(*
SPDX-FileCopyrightText: © 2026 Oleksandr Tiutyk <trofimich@gmail.com>
SPDX-License-Identifier: MIT
License: https://opensource.org/license/mit
*)

(*!
<summary>Provides common automation state, diagnostics and local event reception.</summary>
<description>
Both event delivery directions call OnEventReceived locally. Descendants with a parent or children extend the
appropriate direction with forwarding; terminal nodes only receive the event. Event delivery is synchronous
and borrowed, without retaining the event or transferring ownership. Delivery and forwarding are independent
of Enabled and operational state. OnEventReceived decides whether the component should react in its current
state; inactivity alone does not stop propagation. The event must be non-null and live. Handler exceptions
abort delivery and propagate to the caller; effects of handlers already invoked are not rolled back.
Initialization validates required dependencies before hooks. Child types require a live borrowed parent.
FALSE reports pending initialization or failure; INVALID must never report successful initialization.
Error and HasError observe the same diagnostic selected by GetReportedError(). The base exposes its execution error.
Required error snapshots precede logging callbacks so they preserve the primary diagnostic.
Stop transitions a WORKING component (and, for branches, all WORKING children) to STOPPED regardless of
Enabled, so a runtime stop reaction also stops a disabled working component and preserves its Reset requirement.
</description>
*)

FUNCTION_BLOCK ABSTRACT AutomationComponent EXTENDS TOF_Core.Object IMPLEMENTS IAutomationComponent
VAR
	{attribute 'hide'} 
	_Name : WSTRING;

	{attribute 'hide'} 
	_Enabled : BOOL := TRUE;
	
	{attribute 'hide'} 
	_OperationalState : OPERATIONAL_STATE;
	//! <summary>Counts state transitions so output traversal can detect a stop followed by an immediate reset.</summary>
	_OperationalStateRevision : UDINT;	
	{attribute 'hide'} 
	_OperationalStateReason : WSTRING(255);	

	_InitializationTimer : Tc2_Standard.TON;
	
	{attribute 'hide'} 
	_Error : TOF_Core.ERROR;
	
	{attribute 'hide'} 
	_ExceptionHandlingPolicy : TOF_Core.IExceptionHandlingPolicy;
END_VAR

(*!
<summary>Receives a broadcast event locally without forwarding it.</summary>
<description>
Calls OnEventReceived once. This is the terminal behavior for a leaf; branches override it to forward to
children unless propagation is stopped. Handled does not suppress delivery. The event is borrowed for this
synchronous call and is not retained or owned by the component.
</description>
*)

METHOD BroadcastEvent
VAR_INPUT
	event : TOF_Core.IEvent;
END_VAR
VAR
	stopPropagation : BOOL;
END_VAR
OnEventReceived(event := event, stopPropagation => stopPropagation);
END_METHOD

(*!
<summary>Receives a bubbling event locally without forwarding it.</summary>
<description>
Calls OnEventReceived once. This is the terminal behavior for a root; components with a parent override it to
forward upward unless propagation is stopped. Handled does not suppress delivery. The event is borrowed for
this synchronous call and is not retained or owned by the component.
</description>
*)

METHOD BubbleEvent
VAR_INPUT
	event : TOF_Core.IEvent;
END_VAR
VAR
	stopPropagation : BOOL;
END_VAR
OnEventReceived(event := event, stopPropagation => stopPropagation);
END_METHOD

(*!
<summary>Disables cyclic execution and invokes disable hooks.</summary>
<description>
Branches also disable their children. Hook exceptions propagate to the caller without rolling back prior
effects.
</description>
*)
METHOD ABSTRACT Disable
END_METHOD

(*!
<summary>Enables cyclic execution and invokes enable hooks.</summary>
<description>
Enabling does not automatically reset a STOPPED component; components stopped while disabled or disabled
while stopped remain STOPPED after Enable until explicitly Reset.
</description>
<param name="includeChildren">When TRUE on a branch, recursively enables child components.</param>
*)
METHOD ABSTRACT Enable
VAR_INPUT
	includeChildren : BOOL := TRUE;
END_VAR
END_METHOD

{attribute 'monitoring' := 'call'}
PROPERTY FINAL Enabled : BOOL
GET
Enabled := _Enabled;
END_GET
END_PROPERTY

(*!
<summary>Gets a borrowed view of the currently reported diagnostic.</summary>
<description>
Read the property again after component execution because a descendant can select a different record.
Observe the reference on the owning task while the component is live, following the IErrorProvider contract.
</description>
*)
{attribute 'monitoring' := 'call'}
PROPERTY FINAL Error : REFERENCE TO TOF_Core.ERROR
GET
Error REF= GetReportedError();
END_GET
END_PROPERTY

{attribute 'monitoring' := 'call'}
PROPERTY FINAL ExceptionHandlingPolicy : TOF_Core.IExceptionHandlingPolicy
GET
ExceptionHandlingPolicy := _ExceptionHandlingPolicy;
END_GET
SET
_ExceptionHandlingPolicy := ExceptionHandlingPolicy;
END_SET
END_PROPERTY

METHOD ABSTRACT Execute
END_METHOD

METHOD FB_init : BOOL
VAR_INPUT
	bInitRetains : BOOL; // TRUE: the retain variables are initialized (reset warm / reset cold)
	bInCopyCode : BOOL;  // TRUE: the instance will be copied to the copy code afterward (online change)
	name : WSTRING;
END_VAR
_Name := SEL(
	TOF_Core.WideStrings.IsNullOrWhiteSpace(stringToCheck := name),
	name,
	GetDefaultName()
);
_InitializationTimer.PT := Parameters.InitializationTimeout;
END_METHOD

METHOD FINAL GetEffectiveExceptionHandlingPolicy : TOF_Core.IExceptionHandlingPolicy
VAR
	thisAsChildAutomationComponent : IChildAutomationComponent;
	parent : IParentAutomationComponent;
END_VAR
IF _ExceptionHandlingPolicy <> 0 THEN
	GetEffectiveExceptionHandlingPolicy := _ExceptionHandlingPolicy;
ELSIF __QUERYINTERFACE(THIS^, thisAsChildAutomationComponent) THEN
	parent := thisAsChildAutomationComponent.Parent;

	IF parent <> 0 THEN
		GetEffectiveExceptionHandlingPolicy := parent.GetEffectiveExceptionHandlingPolicy();
	END_IF
END_IF
END_METHOD

METHOD PROTECTED FINAL GetErrorSeverityByExceptionReaction : TOF_Core.ERROR_SEVERITY
VAR_INPUT
	exceptionReaction : TOF_Core.EXCEPTION_REACTION;
END_VAR
IF exceptionReaction = TOF_Core.EXCEPTION_REACTION.SET_ERROR_AND_STOP THEN
	GetErrorSeverityByExceptionReaction := TOF_Core.ERROR_SEVERITY.CRITICAL;
ELSE
	GetErrorSeverityByExceptionReaction := TOF_Core.ERROR_SEVERITY.ERROR;
END_IF
END_METHOD

(*!
<summary>Prepares diagnostic text locally before passing it to read-only logging or exception parameters.</summary>
<description>Computed diagnostic strings are held in local buffers for the duration of the receiving call.</description>
*)
METHOD HandleRequest
VAR_INPUT
	request	: TOF_Core.INamed;
END_VAR
VAR
	formattedLogMessage : TOF_Core.ERROR_MESSAGE;
END_VAR
IF request = 0 THEN
	RETURN;
END_IF

formattedLogMessage := TOF_Core.WideStrings.Concat255("Request ", request.Name, " was not handled");

TOF_Core.LogManager.TryLogMessage(
	message := formattedLogMessage,
	category := TOF_Core.LOG_CATEGORY.INFORMATION,
	topic1 := TO_WSTRING(ClassName),
	topic2 := TO_WSTRING(__POUNAME())
);
END_METHOD

(*!
<summary>Selects the live diagnostic record exposed by Error and HasError.</summary>
<description>
Returns the component's execution record by default. An override must return a valid reference to
instance-owned storage, including when no error is active. Selection must be side-effect free and must
complete without exceptions. Read the selected record on the component's owner task.
</description>
*)
METHOD PROTECTED GetReportedError : REFERENCE TO TOF_Core.ERROR
GetReportedError REF= _Error;
END_METHOD

(*!
<summary>Reports whether the currently selected diagnostic contains an active error.</summary>
*)
{attribute 'monitoring' := 'call'}
PROPERTY FINAL HasError : BOOL
GET
HasError := THIS^.Error.HasError;
END_GET
END_PROPERTY

(*!
<summary>Sets the maximum wait for pending initialization.</summary>
<description>
T#0S selects Parameters.InitializationTimeout immediately upon assignment, so the getter always returns the
active non-zero duration. Branches expand this duration to at least the maximum InitializationTimeout of their
children during initialization.
</description>
*)
{attribute 'monitoring' := 'call'}
PROPERTY FINAL InitializationTimeout : TIME
GET
InitializationTimeout := _InitializationTimer.PT;
END_GET
SET
_InitializationTimer.PT := SEL(
	InitializationTimeout = T#0S,
	InitializationTimeout,
	Parameters.InitializationTimeout
);
END_SET
END_PROPERTY

(*!
<summary>Validates mandatory dependencies and advances initialization.</summary>
<description>
FALSE reports pending work or failure. An INVALID component must never report TRUE. Caught failures
record a critical copied error and enter terminal INVALID. Completed callback effects are not rolled back.
Only a pending call evaluates the timeout. Completion on the deadline cycle succeeds.
</description>
*)
METHOD ABSTRACT Initialize : BOOL
END_METHOD

{attribute 'monitoring' := 'call'}
PROPERTY FINAL Name : REFERENCE TO WSTRING
GET
Name REF= _Name;
END_GET
END_PROPERTY

(*!
<summary>Handles a delivered event locally and can stop further propagation along the current route.</summary>
<description>
May be called regardless of Enabled or operational state, including while disabled or stopped. The handler
checks state when its reaction requires it. Ignoring an event does not stop propagation; leave stopPropagation
FALSE unless further delivery along the route must be stopped. The event must be non-null and live and is
borrowed only for the call; do not retain it for later use. Handled and stopPropagation are independent.
Setting stopPropagation stops bubbling to the parent or broadcasting into this node's descendants; it does not
cancel sibling branches in the caller. An exception aborts delivery and propagates to the dispatch caller,
without rolling back prior effects.
</description>
*)

METHOD OnEventReceived
VAR_INPUT
	event : TOF_Core.IEvent;
END_VAR
VAR_OUTPUT
	stopPropagation : BOOL;
END_VAR
END_METHOD

METHOD PROTECTED FINAL OnHandleException : TOF_Core.EXCEPTION_REACTION
VAR_INPUT
	exception : TOF_Core.IException;
	failedMethodName : STRING(255);
END_VAR
VAR
	effectiveExceptionHandlingPolicy : TOF_Core.IExceptionHandlingPolicy;
END_VAR
effectiveExceptionHandlingPolicy := GetEffectiveExceptionHandlingPolicy();

IF effectiveExceptionHandlingPolicy <> 0 THEN
	OnHandleException := effectiveExceptionHandlingPolicy.HandleException(
		exception := exception,
		handlingObject := THIS^,
		failedMethodName := failedMethodName
	);
ELSE
	OnHandleException := TOF_Core.EXCEPTION_REACTION.SET_ERROR_AND_STOP;
END_IF
END_METHOD

METHOD PROTECTED OnOperationalStateChanged
VAR_INPUT
	previousState : OPERATIONAL_STATE;
END_VAR
END_METHOD

(*!
<summary>Runs at the start of cyclic working execution when clearing a non-critical error.</summary>
<description>
The base implementation does nothing. An exception raised by OnRecover always records a copied CRITICAL
error and stops the component without consulting ExceptionHandlingPolicy.
</description>
*)
METHOD PROTECTED OnRecover
END_METHOD

{attribute 'monitoring' := 'call'}
PROPERTY FINAL OperationalState : OPERATIONAL_STATE
GET
OperationalState := _OperationalState;
END_GET
END_PROPERTY

{attribute 'monitoring' := 'call'}
PROPERTY FINAL OperationalStateReason : REFERENCE TO WSTRING(255)
GET
OperationalStateReason REF= _OperationalStateReason;
END_GET
END_PROPERTY

METHOD PROTECTED ProcessChildError
VAR_INPUT
	childError : REFERENCE TO TOF_Core.ERROR;  
	childErrorReaction : CHILD_CRITICAL_ERROR_REACTION;	
	childErrorSourceHint : WSTRING(255);
END_VAR

IF NOT __ISVALIDREF(childError)
	OR_ELSE childError.Empty
	OR_ELSE childError.Severity <> TOF_Core.ERROR_SEVERITY.CRITICAL
THEN
	RETURN;
END_IF

IF OperationalState <> OPERATIONAL_STATE.INITIALIZING THEN
	CASE childErrorReaction OF
		CHILD_CRITICAL_ERROR_REACTION.SET_ERROR_AND_CONTINUE:
			IF _Error.Empty THEN
				_Error := childError;
				_Error.SetSeverity(severity := TOF_Core.ERROR_SEVERITY.ERROR);
			END_IF		
		
		CHILD_CRITICAL_ERROR_REACTION.SET_ERROR_AND_STOP:
			IF _Error.Empty OR_ELSE _Error.Severity < TOF_Core.ERROR_SEVERITY.CRITICAL THEN
				_Error := childError;
				_Error.SetSeverity(severity := TOF_Core.ERROR_SEVERITY.CRITICAL);
			END_IF	
			
			IF OperationalState = OPERATIONAL_STATE.WORKING THEN
				Stop(reason := childErrorSourceHint);		
			END_IF
	END_CASE
ELSE
	_Error := childError;
	
	SetOperationalState(state := OPERATIONAL_STATE.INVALID, reason := childErrorSourceHint);		
END_IF
END_METHOD

(*!
<summary>Applies an exception reaction to copied diagnostics and operational state.</summary>
<description>
Initialization failures enter INVALID with a critical error. At runtime a stop reaction records a
critical error and calls Stop on a working component, including when disabled (since Stop transitions
WORKING components and WORKING children to STOPPED regardless of Enabled). This preserves the Reset
requirement after a failed disabled service callback. When the reaction requires an error copy, it is
completed before logging callbacks can reuse a task-local exception. Conversion failures may propagate before
logging and state transitions.
</description>
*)
METHOD PROTECTED ProcessException
VAR_INPUT
	exception : TOF_Core.IException;  
	exceptionReaction : TOF_Core.EXCEPTION_REACTION;	
	exceptionSourceHint : WSTRING(255);
END_VAR
IF exception = 0 OR_ELSE exception.Empty THEN
	RETURN;
END_IF

IF OperationalState = OPERATIONAL_STATE.INITIALIZING THEN
	exception.ToError(targetError := _Error, severity := TOF_Core.ERROR_SEVERITY.CRITICAL);
	TOF_Core.LogManager.TryLogException(exception := exception, severity := TOF_Core.ERROR_SEVERITY.CRITICAL);
	SetOperationalState(state := OPERATIONAL_STATE.INVALID, reason := exceptionSourceHint);

	RETURN;
END_IF

CASE exceptionReaction OF
	TOF_Core.EXCEPTION_REACTION.SET_ERROR_AND_CONTINUE:
		IF _Error.Empty THEN
			exception.ToError(targetError := _Error, severity := TOF_Core.ERROR_SEVERITY.ERROR);
		END_IF

	TOF_Core.EXCEPTION_REACTION.SET_ERROR_AND_STOP:
		IF _Error.Empty OR_ELSE _Error.Severity < TOF_Core.ERROR_SEVERITY.CRITICAL THEN
			exception.ToError(targetError := _Error, severity := TOF_Core.ERROR_SEVERITY.CRITICAL);
		END_IF
END_CASE

TOF_Core.LogManager.TryLogException(
	exception := exception,
	severity := GetErrorSeverityByExceptionReaction(exceptionReaction := exceptionReaction)
);

IF exceptionReaction = TOF_Core.EXCEPTION_REACTION.SET_ERROR_AND_STOP
	AND_THEN OperationalState = OPERATIONAL_STATE.WORKING
THEN
	Stop(reason := exceptionSourceHint);
END_IF
END_METHOD

(*!
<summary>Attempts to recover an enabled stopped component to WORKING.</summary>
<description>
Served only while Enabled and STOPPED. Clears the previous error before reset hooks. A failure in the
component's own reset hook always leaves the component STOPPED with a copied CRITICAL error without
consulting ExceptionHandlingPolicy.
</description>
*)
METHOD ABSTRACT Reset
END_METHOD

(*!
<summary>Records the state and reason and notifies descendants on a transition.</summary>
<description>Advances the transition counter before callbacks so an interrupted output pass can be detected.</description>
<param name="state">New operational state.</param>
<param name="reason">Reason recorded even when the state stays the same.</param>
*)
METHOD PROTECTED SetOperationalState
VAR_INPUT
	state : OPERATIONAL_STATE;
	reason : WSTRING(255);
END_VAR
VAR
	previousState : OPERATIONAL_STATE;

	exceptionCode : __SYSTEM.ExceptionCode;
	exception : TOF_Core.IException;
END_VAR
_OperationalStateReason := reason;

IF _OperationalState = state THEN
	RETURN;
END_IF

previousState := _OperationalState;

_OperationalState := state;
_OperationalStateRevision := _OperationalStateRevision + 1;

__TRY
	OnOperationalStateChanged(previousState := previousState);
__CATCH(exceptionCode)
	exception := TOF_Core.ExceptionManager.GetLastException(
		exceptionCode := exceptionCode,
		catchPointNamespaceName := NamespaceName,
		catchPointPOUName := __POUNAME(),
		catchPointPosition := __POSITION()
	);

	TOF_Core.LogManager.TryLogException(
		exception := exception,
		severity := TOF_Core.ERROR_SEVERITY.ERROR,
		topic1 := "AutomationComponent",
		topic2 := "AutomationComponent.OnOperationalStateChanged"
	);
__ENDTRY
END_METHOD

(*!
<summary>Transitions a WORKING component to OPERATIONAL_STATE.STOPPED.</summary>
<description>
Transitions a WORKING component (and, for branches, all WORKING children) to OPERATIONAL_STATE.STOPPED
regardless of Enabled.
</description>
<param name="reason">Descriptive reason stored in OperationalStateReason.</param>
*)
METHOD ABSTRACT Stop
VAR_INPUT
	reason : WSTRING(255) := "External stop";
END_VAR
END_METHOD

END_FUNCTION_BLOCK

(* stored: Version 1.1.0.1
   POU AutomationComponent: Id {b4897826-50fc-4a14-bfab-9ca314d8ba3a}, SpecialFunc None
   Folder Methods to override: Id {9e76983f-3aef-47df-97e1-2bd089a83751}
   Folder Service methods: Id {1ca304da-6558-4606-898c-97a283347ac4}
   Method BroadcastEvent: Id {d67c04d1-58bd-4df7-9b20-74ea96e2adc1}
   Method BubbleEvent: Id {829ca0e6-191f-4c0e-a95b-b8275c1a0d3c}
   Method Disable: Id {0d1971e1-5f59-4975-85f2-7a8ffd650e1f}
   Method Enable: Id {8c41e56c-f727-473a-87e6-57596090402c}
   Property Enabled: Id {aa3b4270-b240-4ce9-898f-afdfb0a11b5d}
   Get Get: Id {cbdce78d-e4f1-4903-acbe-f5f5552fc11c}
   Property Error: Id {5fa83344-3a33-4d67-90ca-8bcde7966cab}
   Get Get: Id {235d8903-5057-4d40-bc79-b2feb6c602fe}
   Property ExceptionHandlingPolicy: Id {e064b9d3-6917-45e3-8d79-01a4add07dcf}
   Get Get: Id {94ab69af-76bc-482e-a529-660a7e83bff5}
   Set Set: Id {aced67c1-ebd6-481b-9292-25eecf0c2d60}
   Method Execute: Id {0c62a304-be7d-4b17-9ec6-dcdf997a75e1}
   Method FB_init: Id {bf2ff865-6631-4d1d-87f4-db36001851c5}
   Method GetEffectiveExceptionHandlingPolicy: Id {a5117f66-8c2d-49d4-b653-6af2e9154e98}
   Method GetErrorSeverityByExceptionReaction: Id {98732844-72c9-4551-a282-65985e6af1f9}
   Method HandleRequest: Id {13aff68a-a752-4191-bc9a-adaacd1893cd}
   Method GetReportedError: Id {b2f085d3-87bf-4ab7-a602-eddf20559631}
   Property HasError: Id {b058a64f-59a4-414d-b578-01945ffe1e29}
   Get Get: Id {eb91f7b0-98b0-4715-8902-1de1214ef783}
   Property InitializationTimeout: Id {9b430821-2485-45c1-aea1-812b2962dbb2}
   Get Get: Id {87c850fb-dc27-4c26-beea-f228fa9042e3}
   Set Set: Id {496bac58-2886-40a5-a9c9-db583b496ce0}
   Method Initialize: Id {dc8b4ac8-c6c4-4b95-8f4f-93a38c521c55}
   Property Name: Id {d5360ad2-87f6-417b-90ba-8dca4c24bf1d}
   Get Get: Id {11c15535-41cd-4e37-8636-f3d89f13858c}
   Method OnEventReceived: Id {f94f2cee-1148-4676-b329-3c117e050581}
   Method OnHandleException: Id {29c90bad-df55-4870-9c1d-40408bd01466}
   Method OnOperationalStateChanged: Id {dd76bd0f-568b-4bbf-812c-974cfb78aee7}
   Method OnRecover: Id {4fd00d17-dbcf-4903-91de-2486b0cb165f}
   Property OperationalState: Id {f3ab473a-80e6-4bd6-b784-752a1cb14670}
   Get Get: Id {7d4b34b5-9ddf-46c0-9b80-9ef6df164cce}
   Property OperationalStateReason: Id {f68dd7cb-5882-4a97-880b-c0e34a9a06a5}
   Get Get: Id {165bb29f-d77b-4b59-a0e9-8113a39adaab}
   Method ProcessChildError: Id {078f9fd6-7339-4d22-92c2-4a63371d65ff}
   Method ProcessException: Id {7e03d0ad-992f-40a8-92de-f216a0c3449a}
   Method Reset: Id {d9e3b1b6-5f1c-4e0c-b7fb-2f75b7f46fbb}
   Method SetOperationalState: Id {5277f682-bec2-4af0-819a-10cc9e1fbd19}
   Method Stop: Id {7d81c2ed-cf1e-4941-91df-b5092c404637} *)
